TYPE ST_MCHMIPrepareScreen_02_XX_IngredientList :
STRUCT
	arrIndegriend			: ARRAY [1..GVL_MCHMIConstans.NUMBER_INDEGRIEND_ON_PAGE] OF ST_BaseHMIDescriptor;
	iSelectedRow			: INT; //numer wybranego składnika
	iSelectedRowPrev		: INT; //numer wybranego składnika - poprzedni
	bSelectedRow			: BOOL;
	
END_STRUCT
END_TYPE

(* stored: Version 1.1.0.1
   DUT ST_MCHMIPrepareScreen_02_XX_IngredientList: Id {e725ee8e-f225-0f50-1dfa-6dbadeac5a6f} *)
